INTERFACE I_DualPositionActuator

METHOD PUBLIC Activate
END_METHOD

METHOD PUBLIC Disable
END_METHOD

METHOD GetDisableTimeoutTime : TIME
END_METHOD

METHOD GetEnableTimeoutTime : TIME
END_METHOD

METHOD GetState : E_DualPositionActuatorState
END_METHOD

METHOD SetDisableTimeoutTime
VAR_INPUT
    tDisableTimeoutTime : TIME;
END_VAR
END_METHOD

METHOD SetEnableTimeoutTime
VAR_INPUT
    tEnableTimeoutTime : TIME;
END_VAR
END_METHOD

END_INTERFACE

(* stored: Version 1.1.0.1, ProductVersion 3.1.4024.12
   Itf I_DualPositionActuator: Id {96153ad2-1837-4ab0-b1c7-7d77b200ef74}
   Method Activate: Id {72b183e9-6057-431e-881e-7e8c84fefbb8}
   Method Disable: Id {0e53722d-dae9-4737-8f61-6bc15d545bfd}
   Method GetDisableTimeoutTime: Id {ea7bef2c-f934-4142-ade7-527178a732da}
   Method GetEnableTimeoutTime: Id {bc94750c-191f-41f8-89a6-fb42e1e32b35}
   Method GetState: Id {2421db97-9733-4383-a8ba-a03ff838cfce}
   Method SetDisableTimeoutTime: Id {21ca87ac-6962-447d-b832-7d7c60e0562f}
   Method SetEnableTimeoutTime: Id {9aaf12a8-12a0-47af-89b0-8efea9626225} *)
